{attribute addProperty BoxType "EPP2316-0003-0016"}
{attribute addProperty Id "Safe_state_activeAT %I*BOOL811Error_channelAT %I*ARRAY[0 ..1] OF BOOL1620Sync_errorAT %I*BOOL8132TxPDO_ToggleAT %I*BOOL819"}
{attribute addProperty CRC "216293427"}
{attribute addProperty SizeInBites "40"}
{attribute addProperty SizeInBytes "5"}
TYPE DIG_Inputs_Device_30BACB40 :
STRUCT
	{attribute addProperty Name "Safe_state_active"}
	Safe_state_active AT %I* : BOOL;
	{attribute addProperty Name "Error_channel"}
	Error_channel AT %I* : ARRAY[0 ..1] OF BOOL;
	{attribute addProperty Name "Sync_error"}
	Sync_error AT %I* : BOOL;
	{attribute addProperty Name "TxPDO_Toggle"}
	TxPDO_Toggle AT %I* : BOOL;
END_STRUCT
END_TYPE

(* stored: Version 1.2.0.0, ProductVersion 3.1.4024.9
   DUT DIG_Inputs_Device_30BACB40: Id {b1f40f71-a663-4d06-b2cf-d756388fb984} *)
